// TwinCAT 3 PLC project Plc
// ProgramVersion: 3.1.4024.0
// libraries:
//   Tc2_Standard, * (Beckhoff Automation GmbH)
//   Tc2_System, * (Beckhoff Automation GmbH)
//   Tc3_EventLogger, * (Beckhoff Automation GmbH)
//   Tc3_Module, * (Beckhoff Automation GmbH)
// project tree:
//   DUTs/ ST_MyStruct.TcDUT, ST_Point.TcPOU
//   / PlcTask.TcTTO
//   POUs/ AlargEx.TcPOU, Alarming.TcPOU, AlarmingEx.TcPOU, LineChart_Old.TcPOU, MAIN.TcPOU
// real-time tasks:
//   TASK PlcTask: cycle T#10ms, priority 20, ADS port 350

CONFIGURATION Plc
    RESOURCE PLC ON TwinCAT3
        TASK PlcTask(INTERVAL := T#10ms, PRIORITY := 20);
        PROGRAM MAIN WITH PlcTask : MAIN;
    END_RESOURCE
END_CONFIGURATION

// ---- DUTs/ST_MyStruct.TcDUT
TYPE ST_MyStruct :
STRUCT
	xxxx	: INT;
	yyyy	: INT;
END_STRUCT
END_TYPE

// ---- POUs/MAIN.TcPOU
PROGRAM MAIN
VAR
	iCounter : INT;
	bToggle: BOOL;
	bReset: BOOL;
	stext : STRING := 'Start';
	
	
	fbAlarmingEx	: AlarmingEx;
	
	bAlarm 		: BOOL;
	iAlarm		: INT;
	
	stStruct1		: ST_MyStruct;
	
	arrData			: ARRAY[0..99] OF INT;
bInit				: BOOL := TRUE;
	i: INT;
END_VAR

IF bInit THEN
	bInit := FALSE;
	FOR i:=0 TO 99 DO
		arrData[i] := (i MOD 20);
	END_FOR
END_IF
LineChart_Old();


IF bToggle THEN
	iCounter := (iCounter+1 ) MOD 1000;
	sText := 'Start';
	IF iCounter = 0 THEN
		bToggle := FALSE;
	END_IF
ELSE
	sText := 'Stop';
	(*
	IF bReset THEN
		bReset := FALSE;
		iCounter := 0;
	END_IF*)

END_IF

Alarming();
fbAlarmingEx();

END_PROGRAM

// ---- POUs/AlarmingEx.TcPOU
FUNCTION_BLOCK AlarmingEx
VAR_INPUT
END_VAR
VAR_OUTPUT
END_VAR
VAR
	bInit			: BOOL := TRUE;
	bRaise			: BOOL;
	bClear			: BOOL;
	
	fbAlm			: FB_TcAlarm;
	fbSourceInfo	: FB_TcSourceInfo;
END_VAR

IF bInit THEN
	bInit := FALSE;
	
	fbSourceInfo.Clear();
	fbSourceInfo.sName := '%l%L_MyName%/l%';
	
	//fbAlm.CreateEx(TC_Events.MyEventClass.MyAlarm, TRUE, 0);
	fbAlm.CreateEx(TC_Events.MyEventClass.MyFirstAlarm, TRUE, fbSourceInfo);
	
	fbAlm.ipArguments.Clear();
	fbAlm.ipArguments.AddString('BMK');
END_IF


IF bClear AND (fbAlm.eConfirmationState = TcEventConfirmationState.Confirmed) THEN
	bClear := FALSE;
	fbAlm.Clear(0, FALSE);
END_IF

{attribute 'TcRpcEnable'}
METHOD RaiseAlarm : BOOL
VAR_INPUT
END_VAR
fbAlm.Raise(0);
END_METHOD

END_FUNCTION_BLOCK

// ---- POUs/LineChart_Old.TcPOU
PROGRAM LineChart_Old
VAR
	aPoints : ARRAY [1..2,1..100] OF ST_Point;
	
	bInit : BOOL := TRUE;
	nCounter: INT;
	nValue1 : INT := 1;
	nValue2 : INT := -1;
END_VAR

IF bInit THEN
	FOR nCounter := 1 TO 100 DO
		aPoints[1, nCounter].x := nCounter;
		aPoints[2, nCounter].x := nCounter;
		aPoints[2, nCounter].y := 100;
	END_FOR
	
	bInit := FALSE;
END_IF

// graph 1
FOR nCounter := 100 TO 2 BY -1 DO
	aPoints[1, nCounter].y := aPoints[1, nCounter - 1].y;
END_FOR

aPoints[1, 1].y := aPoints[1, 1].y + nValue1;

IF aPoints[1, 1].y = 100 THEN
	nValue1 := -1;
ELSIF aPoints[1, 1].y = 1 THEN
	nValue1 := 1;
END_IF 

// graph 2
FOR nCounter := 100 TO 2 BY -1 DO
	aPoints[2, nCounter].y := aPoints[2, nCounter - 1].y;
END_FOR

aPoints[2, 1].y := aPoints[2, 1].y + nValue2;

IF aPoints[2, 1].y = 100 THEN
	nValue2 := -1;
ELSIF aPoints[2, 1].y = 1 THEN
	nValue2 := 1;
END_IF

END_PROGRAM

// ---- DUTs/ST_Point.TcPOU
TYPE ST_Point :
STRUCT
	x : INT;
	y : INT;
END_STRUCT
END_TYPE

// ---- POUs/Alarming.TcPOU
PROGRAM Alarming
VAR
	bInit	: BOOL := TRUE;
	bSend	: BOOL;

	fbMsg	: FB_TcMessage;
END_VAR

IF bInit THEN
	bInit := FALSE;
	fbMsg.CreateEx(TC_EVENTS.MyEventClass.MyFirstMessage, 0);
END_IF

IF bSend THEN
	bSend := FALSE;
	fbMsg.Send(0);
END_IF

END_PROGRAM

// ---- POUs/AlargEx.TcPOU
PROGRAM AlargEx
VAR
	bInit			: BOOL := TRUE;
	bRaise			: BOOL;
	bClear			: BOOL;
	
	fbAlm			: FB_TcAlarm;
	fbSourceInfo	: FB_TcSourceInfo;
END_VAR

IF bInit THEN
	bInit := FALSE;
	
	fbSourceInfo.Clear();
	fbSourceInfo.sName := '%l%L_MyName%/l%';
	
	//fbAlm.CreateEx(TC_Events.MyEventClass.MyAlarm, TRUE, 0);
	fbAlm.CreateEx(TC_Events.MyEventClass.MyFirstAlarm, TRUE, fbSourceInfo);
	
	fbAlm.ipArguments.Clear();
	fbAlm.ipArguments.AddString('BMK');
END_IF

IF bRaise THEN
	bRaise := FALSE;
	fbAlm.Raise(0);
END_IF

IF bClear AND (fbAlm.eConfirmationState = TcEventConfirmationState.Confirmed) THEN
	bClear := FALSE;
	fbAlm.Clear(0, FALSE);
END_IF

END_PROGRAM
